// TIA Portal V18 export
DATA_BLOCK "DB_CLOUD_Simulation"   // DB1200
{ S7_Optimized_Access := 'FALSE' }
VERSION : 0.1
// stored: AutoNumber false, DBAccessibleFromOPCUA true, DBAccessibleFromWebserver true, IsOnlyStoredInLoadMemory false, IsWriteProtectedInAS false
   VAR RETAIN
      Array_1 : Array[1..90] of Real;
      P1S1CO2 : Real := 0.0;
      P1S1MT : Real := 1.0;
      P1S1H : Real := 2.0;
      P1S1PH : Real := 3.0;
      P1S2O2 : Real := 4.0;
      P1S2CO2 : Real := 5.0;
      P1S2MT : Real := 6.0;
      P1S2H : Real := 7.0;
      P1S2PH : Real := 8.0;
      P1S3O2 : Real := 9.0;
      P1S3CO2 : Real := 10.0;
      P1S3MT : Real := 11.0;
      P1S3H : Real := 12.0;
      P1S3PH : Real := 13.0;
      P2S1O2 : Real := 14.0;
      P2S1CO2 : Real := 15.0;
      P2S1MT : Real := 16.0;
      P2S1H : Real := 17.0;
      P2S1PH : Real := 18.0;
      P2S2O2 : Real := 19.0;
      P2S2CO2 : Real := 20.0;
      P2S2MT : Real := 21.0;
      P2S2H : Real := 22.0;
      P2S2PH : Real := 23.0;
      P2S3O2 : Real := 24.0;
      P2S3CO2 : Real := 25.0;
      P2S3MT : Real := 26.0;
      P2S3H : Real := 27.0;
      P2S3PH : Real := 28.0;
      P3S1O2 : Real := 29.0;
      P3S1CO2 : Real := 30.0;
      P3S1MT : Real := 31.0;
      P3S1H : Real := 32.0;
      P3S1PH : Real := 33.0;
      P3S2O2 : Real := 34.0;
      P3S2CO2 : Real := 35.0;
      P3S2MT : Real := 36.0;
      P3S2H : Real := 37.0;
      P3S2PH : Real := 38.0;
      P3S3O2 : Real := 39.0;
      P3S3CO2 : Real := 40.0;
      P3S3MT : Real := 41.0;
      P3S3H : Real := 42.0;
      P3S3PH : Real := 43.0;
      P4S1O2 : Real := 44.0;
      P4S1CO2 : Real := 45.0;
      P4S1MT : Real := 46.0;
      P4S1H : Real := 47.0;
      P4S1PH : Real := 48.0;
      P4S2O2 : Real := 49.0;
      P4S2CO2 : Real := 50.0;
      P4S2MT : Real := 51.0;
      P4S2H : Real := 52.0;
      P4S2PH : Real := 53.0;
      P4S3O2 : Real := 54.0;
      P4S3CO2 : Real := 55.0;
      P4S3MT : Real := 56.0;
      P4S3H : Real := 57.0;
      P4S3PH : Real := 58.0;
      P5S1O2 : Real := 59.0;
      P5S1CO2 : Real := 60.0;
      P5S1MT : Real := 61.0;
      P5S1H : Real := 62.0;
      P5S1PH : Real := 63.0;
      P5S2O2 : Real := 64.0;
      P5S2CO2 : Real := 65.0;
      P5S2MT : Real := 66.0;
      P5S2H : Real := 67.0;
      P5S2PH : Real := 68.0;
      P5S3O2 : Real := 69.0;
      P5S3CO2 : Real := 70.0;
      P5S3MT : Real := 71.0;
      P5S3H : Real := 72.0;
      P5S3PH : Real := 73.0;
      P6S1O2 : Real := 74.0;
      P6S1CO2 : Real := 75.0;
      P6S1MT : Real := 76.0;
      P6S1H : Real := 77.0;
      P6S1PH : Real := 78.0;
      P6S2O2 : Real := 79.0;
      P6S2CO2 : Real := 80.0;
      P6S2MT : Real := 81.0;
      P6S2H : Real := 82.0;
      P6S2PH : Real := 83.0;
      P6S3O2 : Real := 84.0;
      P6S3CO2 : Real := 85.0;
      P6S3MT : Real := 86.0;
      P6S3H : Real := 87.0;
      P6S3PH : Real := 88.0;
   END_VAR
BEGIN
   Array_1[1] := 0.0;
   Array_1[2] := 1.0;
   Array_1[3] := 2.0;
   Array_1[4] := 3.0;
   Array_1[5] := 4.0;
   Array_1[6] := 5.0;
   Array_1[7] := 6.0;
   Array_1[8] := 7.0;
   Array_1[9] := 8.0;
   Array_1[10] := 9.0;
   Array_1[11] := 10.0;
   Array_1[12] := 11.0;
   Array_1[13] := 12.0;
   Array_1[14] := 13.0;
   Array_1[15] := 14.0;
   Array_1[16] := 15.0;
   Array_1[17] := 16.0;
   Array_1[18] := 17.0;
   Array_1[19] := 18.0;
   Array_1[20] := 19.0;
   Array_1[21] := 20.0;
   Array_1[22] := 21.0;
   Array_1[23] := 22.0;
   Array_1[24] := 23.0;
   Array_1[25] := 24.0;
   Array_1[26] := 25.0;
   Array_1[27] := 26.0;
   Array_1[28] := 27.0;
   Array_1[29] := 28.0;
   Array_1[30] := 29.0;
   Array_1[31] := 30.0;
   Array_1[32] := 31.0;
   Array_1[33] := 32.0;
   Array_1[34] := 33.0;
   Array_1[35] := 34.0;
   Array_1[36] := 35.0;
   Array_1[37] := 36.0;
   Array_1[38] := 37.0;
   Array_1[39] := 38.0;
   Array_1[40] := 39.0;
   Array_1[41] := 40.0;
   Array_1[42] := 41.0;
   Array_1[43] := 42.0;
   Array_1[44] := 43.0;
   Array_1[45] := 44.0;
   Array_1[46] := 45.0;
   Array_1[47] := 46.0;
   Array_1[48] := 47.0;
   Array_1[49] := 48.0;
   Array_1[50] := 49.0;
   Array_1[51] := 50.0;
   Array_1[52] := 51.0;
   Array_1[53] := 52.0;
   Array_1[54] := 53.0;
   Array_1[55] := 54.0;
   Array_1[56] := 55.0;
   Array_1[57] := 56.0;
   Array_1[58] := 57.0;
   Array_1[59] := 58.0;
   Array_1[60] := 59.0;
   Array_1[61] := 60.0;
   Array_1[62] := 61.0;
   Array_1[63] := 62.0;
   Array_1[64] := 63.0;
   Array_1[65] := 64.0;
   Array_1[66] := 65.0;
   Array_1[67] := 66.0;
   Array_1[68] := 67.0;
   Array_1[69] := 68.0;
   Array_1[70] := 69.0;
   Array_1[71] := 70.0;
   Array_1[72] := 71.0;
   Array_1[73] := 72.0;
   Array_1[74] := 73.0;
   Array_1[75] := 74.0;
   Array_1[76] := 75.0;
   Array_1[77] := 76.0;
   Array_1[78] := 77.0;
   Array_1[79] := 78.0;
   Array_1[80] := 79.0;
   Array_1[81] := 80.0;
   Array_1[82] := 81.0;
   Array_1[83] := 82.0;
   Array_1[84] := 83.0;
   Array_1[85] := 84.0;
   Array_1[86] := 85.0;
   Array_1[87] := 86.0;
   Array_1[88] := 87.0;
   Array_1[89] := 88.0;
   Array_1[90] := 89.0;
END_DATA_BLOCK
